{attribute 'GeneratedUsingTerminal: EL7342-0000-0023'}
{attribute addProperty BoxType "EL7342-0000-0023"}
{attribute addProperty Id "ControlAT %Q*Control_4AE59EC24"}
{attribute addProperty CRC "2495602655"}
{attribute addProperty Size "4"}
TYPE DCM_Control_Channel_94BFDFDF EXTENDS OutputBase_10CEE7DE :
STRUCT
	{attribute addProperty Name "Control"}
	Control AT %Q* : Control_4AE59EC2;
END_STRUCT
END_TYPE

(* stored: Version 1.2.0.0, ProductVersion 3.1.4024.11
   DUT DCM_Control_Channel_94BFDFDF: Id {2d613371-ecdf-41f0-a773-5fd126ffdf50} *)
